// TIA Portal V17 export
// export: Created 2022-06-16T09:21:08.0209505Z, ExportSetting WithDefaults, DisplayName Totally Integrated Automation Portal, DisplayVersion V17, DisplayName TIA Portal Openness, DisplayVersion V17, DisplayName TIA Portal Version Control Interface, DisplayVersion V17, DisplayName STEP 7 Professional, DisplayVersion V17, DisplayName STEP 7 Safety, DisplayVersion V17, DisplayName WinCC Advanced, DisplayVersion V17
TYPE "typeSatParam"
// stored: IsFailsafeCompliant false
   STRUCT
      deltaSatGainNeg : Real;
      deltaSatGainPos : Real;
      satLevels : Array[1.."AXIS_NUM"] of Real;
   END_STRUCT;
END_TYPE
